{attribute 'GeneratedUsingTerminal: AT2041-0250-0021'}
{attribute addProperty BoxType "AT2041-0250-0021"}
{attribute addProperty Id "A_0101_AT2041_5250_0018_AT2041_5250AT2041_33A3DF1B80"}
{attribute addProperty CRC "2852468728"}
{attribute addProperty Size "80"}
TYPE A_0043_AT2041_0250_0021_AA0537F8 EXTENDS AT2041_2EA6C9BF :
STRUCT
	{attribute addProperty Name "A_0101(AT2041-5250-0018) (AT2041-5250)"}
	{attribute addProperty PreviousPort "A_0043(AT2041-0250-0021) : B"}
	A_0101_AT2041_5250_0018_AT2041_5250 : AT2041_33A3DF1B;
END_STRUCT
END_TYPE

(* stored: Version 1.2.0.0, ProductVersion 3.1.4024.9
   DUT A_0043_AT2041_0250_0021_AA0537F8: Id {2e00d7d0-de83-4862-ad31-bc1c282299fb} *)
